Fanuc KAREL source: kt00918.KL

-- PROVISIONAL review KL for V1013-1; original PC SHA256 995160c5ae8f763b98d3ffd6d19eaff4180e44c598961b8f66de4faaafeb3225
-- Incomplete behavior may be omitted. Consult companion uncertainty JSON. Do not deploy.
PROGRAM KT00918
%NOLOCKGROUP
VAR
  S1 : STRING[80]
  S2 : STRING[80]
  OUT : INTEGER
BEGIN
  -- UNRESOLVED_PC offsets 5-14; opcodes 3F,75
  -- UNRESOLVED_PC offsets 19-28; opcodes 3F,75
  -- UNRESOLVED_PC offsets 33-42; opcodes 3F,75
  -- UNRESOLVED_PC offsets 47-56; opcodes 3F,75
  -- UNRESOLVED_PC offsets 61-86; opcodes 27,22,2A,22,2A,76,23
  -- UNRESOLVED_PC offsets 91-95; opcodes 7F
END KT00918
